{attribute 'linkalways'} 
{attribute 'no_explicit_call' := 'This FB is a CLASS and must be accessed using methods or properties'}
{attribute 'enable_dynamic_creation'}
FUNCTION_BLOCK FINAL AND_INT EXTENDS Node
VAR
	in1 : _INT(0);
	in2 : _INT(0);
	out : _INT(0);
END_VAR

METHOD PUBLIC Clone : I_Node
VAR
	pNode : POINTER TO AND_INT;
END_VAR
pNode := __NEW(AND_INT);
Clone := pNode^;
END_METHOD

METHOD FB_init : BOOL
VAR_INPUT
	bInitRetains : BOOL; // if TRUE, the retain variables are initialized (warm start / cold start)
	bInCopyCode : BOOL;  // if TRUE, the instance afterwards gets moved into the copy code (online change)
END_VAR
AddInput('in1',THIS^.in1);
AddInput('in2',THIS^.in2);
AddOutput('out', THIS^.out);
END_METHOD

METHOD PROTECTED OnExecute
VAR
END_VAR
out.Value := in1.Value AND in2.Value;
END_METHOD

END_FUNCTION_BLOCK

(* stored: Version 1.1.0.1, ProductVersion 3.1.4024.15
   POU AND_INT: Id {6fe323e7-163b-4602-bb6d-48a904b953ff}, SpecialFunc None
   Folder Constructor: Id {83d68aa1-bd26-4c8e-97cf-e36403295f9f}
   Method Clone: Id {54cbcc8d-8a08-4439-a896-0ffb0499f8c8}
   Method FB_init: Id {f8e60ba2-6b2f-4cc4-b6b2-61ee620785f5}
   Method OnExecute: Id {b74c57d6-5da6-44e0-901b-0eaf129d9d55} *)
